FUNCTION F_DCTIME64_TO_ULINT : ULINT
VAR_INPUT
	in:		T_DCTIME64;
END_VAR
VAR
	out:	ULINT;
END_VAR

memcpy (ADR(out), ADR(in), SIZEOF(in));
F_DCTIME64_TO_ULINT	:= out;

END_FUNCTION

(* stored: Version 1.1.0.1, ProductVersion 3.1.4022.9
   POU F_DCTIME64_TO_ULINT: Id {617164a4-8903-46f9-a31d-a20873d167db}, SpecialFunc None *)
